FUNCTION F_FBNameFromPath : STRING // distills .fb name from function path
VAR_INPUT
	sPath	: STRING ;
END_VAR
VAR
	sTemp		: STRING ;
	nstartFbName: INT ; 
END_VAR

sTemp := sPath ;

REPEAT 
	// Look for first occurance of .fb in string
	nStartFbName := FIND( sTemp,'.fb');
	// Delete text before .fb and .fb itself
	IF nstartFbName <>0 THEN 
		sTemp := DELETE( STR := sTemp, LEN := nstartFbName + 3, 0); 
	END_IF
UNTIL
	nstartFbName = 0 
END_REPEAT

F_FBNameFromPath := sTemp ;

END_FUNCTION

(* stored: Version 1.1.0.1, ProductVersion 3.1.4024.4
   POU F_FBNameFromPath: Id {5ade0010-a24a-4a30-b048-09fb95415f37}, SpecialFunc None *)
